// TIA Portal V20 export
DATA_BLOCK "SBK05"   // DB318
// stored: MemoryReserve 100
   VAR
      "GATE EC U/W TOP PB.LOCK" : Bool := FALSE;
      "GATE EC U/W TOP PB.RESET" : Bool := FALSE;
      SPARE : Bool := FALSE;
      SPARE_1 : Bool := FALSE;
      "GATE EC U/W TOP PB.UNLOCK" : Bool := FALSE;
      SPARE_2 : Bool := FALSE;
      SPARE_3 : Bool := FALSE;
      SPARE_4 : Bool := FALSE;
      "GATE EC U/W TOP PL.LOCK" : Bool := TRUE;
      "GATE EC U/W TOP PL.UNLOCK" : Bool := FALSE;
      "GATE EC U/W TOP PL.RESET" : Bool := TRUE;
   END_VAR
BEGIN
END_DATA_BLOCK
